Universal Robots PolyScope program: turco2.urp

Program turco2 (installation=default directory=/programs/usbdisk createdIn=3.15.3.106223 lastSavedIn=3.15.3.106223 robotSerialNumber=2017357015)
Calibrated DH parameters: a=[0.000021, -0.261063, -0.376363, 0.000077, 0.000104, 0]; d=[0.089312, 121.214456, -102.904559, -18.199769, 0.094928, 0.082537]; alpha=[1.569843, -0.002771, -0.006062, 1.56958, -1.570059, 0]; deltaTheta=[0.000006, -0.909999, 0.623282, 0.286705, -0.000096, 0.00002]
InitVariablesNode
BeforeStart
  MoveJ speed 60 deg/s, acceleration 80 deg/s^2 (useActiveTCP=true)
    Waypoint Waypoint_2: TCP in base x=74.543 y=-607.557 z=480.397 mm, rx=3.1317 ry=-0.001 rz=-0.01 rad; joints [-72.397, -119.802, -18.875, -130.938, 89.067, -162.266] deg; flange x=75.658 y=-607.522 z=634.946 mm, rx=3.1317 ry=-0.001 rz=-0.01 rad
  pos_foto := Waypoint_2
  Set ExpressionOutput pin=saida_botao; expression=0
  Set ExpressionOutput pin=mov_feito; expression=0
Robot Program (runOnlyOnce=false)
  If digital_in[0]≟ True
    Set ExpressionOutput pin=saida_botao; expression=1
    Set ExpressionOutput pin=mov_feito; expression=0
    Loop While (checkContinuously=false) expression=saida_botao≟1
      If pode_movimentar≟1
        Call mover_peça
      ElseIf pode_movimentar≟2
        Call captura_peça
      ElseIf pode_movimentar≟3
        Call mover_peça
        Wait Sleep waitTime=1
        Set ExpressionOutput pin=mov_feito; expression=0
        Call mover_peça
SubProgram -> mover_peça
SubProgram -> captura_peça
Thread Thread_1 (runOnlyOnce=false)
  If led≟0
    Set DigitalOutput pin=digital_out[0]; digitalValue=0
    Set DigitalOutput pin=digital_out[1]; digitalValue=0
  ElseIf led≟1
    Set DigitalOutput pin=digital_out[0]; digitalValue=1
    Set DigitalOutput pin=digital_out[1]; digitalValue=0
  ElseIf led≟2
    Set DigitalOutput pin=digital_out[1]; digitalValue=1
    Set DigitalOutput pin=digital_out[0]; digitalValue=0
SubProgram mover_peça (keepSynchronizedWithDisk=false)
  Set DigitalOutput pin=digital_out[0]; digitalValue=1
  x_1 := x_inicial
  x_2 := x_final
  y_1 := y_inicial
  y_2 := y_final
  Set ExpressionOutput pin=saida_botao; expression=0
  ref := get_actual_tcp_pose()
  offset_pega1 := p[x_1/1000,y_1/1000,0,ref[3],ref[4],ref[5]]
  offset_pega2 := p[x_1/1000,y_1/1000,-0.122,ref[3],ref[4],ref[5]]
  offset_solta := p[x_2/1000,y_2/1000,0,ref[3],ref[4],ref[5]]
  offset_solta2 := p[x_2/1000,y_2/1000,-0.122,ref[3],ref[4],ref[5]]
  Set DigitalOutput pin=tool_out[1]; digitalValue=1
  Set DigitalOutput pin=tool_out[0]; digitalValue=0
  MoveL speed 250 mm/s, acceleration 1200 mm/s^2 (useActiveTCP=true) feature=Plane_4
    Waypoint Waypoint (Variable): variable=offset_pega1
    Waypoint Waypoint (Variable): variable=offset_pega2
    Wait Sleep waitTime=0.7
  Set DigitalOutput pin=tool_out[1]; digitalValue=0
  Set DigitalOutput pin=tool_out[0]; digitalValue=1
  Wait Sleep waitTime=0.7
  MoveL speed 250 mm/s, acceleration 1200 mm/s^2 (useActiveTCP=true) feature=Plane_4
    Waypoint Waypoint (Variable): variable=offset_pega1
    Waypoint Waypoint (Variable): variable=offset_solta
    Waypoint Waypoint (Variable): variable=offset_solta2
  Set DigitalOutput pin=tool_out[0]; digitalValue=0
  Set DigitalOutput pin=tool_out[1]; digitalValue=1
  Wait Sleep waitTime=0.7
  MoveL speed 250 mm/s, acceleration 1200 mm/s^2 (useActiveTCP=true) feature=Plane_4
    Waypoint Waypoint (Variable): variable=offset_solta
  Set DigitalOutput pin=digital_out[0]; digitalValue=0
  Set ExpressionOutput pin=mov_feito; expression=1
  MoveJ speed 60 deg/s, acceleration 80 deg/s^2 (useActiveTCP=true)
    Waypoint Waypoint_2: TCP in base x=74.543 y=-607.557 z=480.397 mm, rx=3.1317 ry=-0.001 rz=-0.01 rad; joints [-72.397, -119.802, -18.875, -130.938, 89.067, -162.266] deg; flange x=75.658 y=-607.522 z=634.946 mm, rx=3.1317 ry=-0.001 rz=-0.01 rad
SubProgram captura_peça (keepSynchronizedWithDisk=false)
  Set DigitalOutput pin=digital_out[0]; digitalValue=1
  Set ExpressionOutput pin=saida_botao; expression=0
  x_d := x_descarte
  y_d := y_descarte
  x_1 := x_inicial
  x_2 := x_final
  y_1 := y_inicial
  y_2 := y_final
  ref := get_actual_tcp_pose()
  offset_pega1 := p[x_1/1000,y_1/1000,0,ref[3],ref[4],ref[5]]
  offset_pega2 := p[x_1/1000,y_1/1000,-0.123,ref[3],ref[4],ref[5]]
  offset_solta := p[x_2/1000,y_2/1000,0,ref[3],ref[4],ref[5]]
  offset_solta2 := p[x_2/1000,y_2/1000,-0.123,ref[3],ref[4],ref[5]]
  pos_descarte := p[-x_d/1000,y_d/1000,0,ref[3],ref[4],ref[5]]
  pos_descarte2 := p[-x_d/1000,y_d/1000,-0.118,ref[3],ref[4],ref[5]]
  Set DigitalOutput pin=tool_out[1]; digitalValue=1
  Set DigitalOutput pin=tool_out[0]; digitalValue=0
  MoveL speed 250 mm/s, acceleration 1200 mm/s^2 (useActiveTCP=true) feature=Plane_4
    Waypoint Waypoint (Variable): variable=offset_solta
    Waypoint Waypoint (Variable): variable=offset_solta2
    Set DigitalOutput pin=tool_out[1]; digitalValue=0
    Set DigitalOutput pin=tool_out[0]; digitalValue=1
    Wait Sleep waitTime=0.7
    Waypoint Waypoint (Variable): variable=offset_solta
    Waypoint Waypoint (Variable): variable=pos_descarte
    Waypoint Waypoint (Variable): variable=pos_descarte2
    Set DigitalOutput pin=tool_out[0]; digitalValue=0
    Set DigitalOutput pin=tool_out[1]; digitalValue=1
    Wait Sleep waitTime=0.7
    Waypoint Waypoint (Variable): variable=pos_descarte
    Waypoint Waypoint (Variable): variable=offset_pega1
    Waypoint Waypoint (Variable): variable=offset_pega2
    Set DigitalOutput pin=tool_out[1]; digitalValue=0
    Set DigitalOutput pin=tool_out[0]; digitalValue=1
    Wait Sleep waitTime=0.7
    Waypoint Waypoint (Variable): variable=offset_pega1
    Waypoint Waypoint (Variable): variable=offset_solta
    Waypoint Waypoint (Variable): variable=offset_solta2
    Set DigitalOutput pin=tool_out[0]; digitalValue=0
    Set DigitalOutput pin=tool_out[1]; digitalValue=1
    Wait Sleep waitTime=0.7
    Waypoint Waypoint (Variable): variable=offset_solta
  Set DigitalOutput pin=digital_out[0]; digitalValue=0
  Set ExpressionOutput pin=mov_feito; expression=1
  MoveJ speed 60 deg/s, acceleration 80 deg/s^2 (useActiveTCP=true)
    Waypoint Waypoint_2 referenceName=Waypoint_2: TCP in base x=74.543 y=-607.557 z=480.397 mm, rx=3.1317 ry=-0.001 rz=-0.01 rad; joints [-72.397, -119.802, -18.875, -130.938, 89.067, -162.266] deg; flange x=75.658 y=-607.522 z=634.946 mm, rx=3.1317 ry=-0.001 rz=-0.01 rad
